PROGRAM PRG_SP2K2_TXAS
VAR
	bInit : BOOL := TRUE;
    fbTXAS_TAR_RX : FB_MotionStage;
END_VAR


IF bInit THEN
    Main.M38.bHardwareEnable := TRUE;
    Main.M38.bPowerSelf := TRUE;
    bInit := FALSE;
END_IF


fbTXAS_TAR_RX(stMotionStage:=Main.M38);

END_PROGRAM

(* stored: Version 1.1.0.1, ProductVersion 3.1.4024.12
   POU PRG_SP2K2_TXAS: Id {5d1de4e6-8549-48db-a26e-02c10173afc0}, SpecialFunc None *)
